{attribute 'GeneratedUsingTerminal: AX8108-0100-0101-0101'}
{attribute addProperty BoxType "AX8108-0100-0101-0101"}
{attribute addProperty Id "Std_InputBOOL1Std_Input_1BOOL1Std_Input_2BOOL1Std_Input_3BOOL1Std_Input_4BOOL1Std_Input_5BOOL1Std_Input_6BOOL1Std_Input_7BOOL1"}
{attribute addProperty CRC "1009339169"}
{attribute addProperty Size "8"}
TYPE FSOE_3C294B21 :
STRUCT
	{attribute addProperty Name "Std_Input"}
	Std_Input : BOOL;
	{attribute addProperty Name "Std_Input_1"}
	Std_Input_1 : BOOL;
	{attribute addProperty Name "Std_Input_2"}
	Std_Input_2 : BOOL;
	{attribute addProperty Name "Std_Input_3"}
	Std_Input_3 : BOOL;
	{attribute addProperty Name "Std_Input_4"}
	Std_Input_4 : BOOL;
	{attribute addProperty Name "Std_Input_5"}
	Std_Input_5 : BOOL;
	{attribute addProperty Name "Std_Input_6"}
	Std_Input_6 : BOOL;
	{attribute addProperty Name "Std_Input_7"}
	Std_Input_7 : BOOL;
END_STRUCT
END_TYPE

(* stored: Version 1.2.0.0, ProductVersion 3.1.4024.9
   DUT FSOE_3C294B21: Id {c78ea9d8-ae66-4d83-86b4-2877d75871d2} *)
